FUNCTION_BLOCK Test_TStreamAdd_Read_LINT EXTENDS T_UnitTestBase
VAR
    Stream  : T_Stream(StreamLength := 2);
    ArgType : E_ArgTypeId := E_ArgTypeId.Type_LINT;
END_VAR

METHOD  Init
VAR_INPUT
END_VAR
END_METHOD

{attribute 'analysis' := '-33'} // inhibit unused variable warning
METHOD RunTest
Stream.Init(2);

// add a LINT...
Stream.SetNextArgTypeId(ArgType);
Stream.Add_LINT(123456789);

Stream.SetReadPosition(0);

// check next arg type is correct...
AssertEquals_INT(Expected     := ArgType,
                           Actual       := Stream.GetNextArgTypeId(),
                           Message := 'Stream.GetNextArgTypeId()');

// check next value...	
AssertEquals_LINT(Expected     := 123456789,
                            Actual       := Stream.Read_LINT(),
                            Message := 'Stream.Read_LINT()');

// check we are at the end of the stream..							
AssertEquals_UDINT(Expected     := Stream.StreamLength,
                             Actual       := Stream.ReadPosition,
                             Message := 'Stream.ReadPosition');

TestCompleted := TRUE;
END_METHOD

END_FUNCTION_BLOCK

(* stored: Version 1.1.0.1, ProductVersion 3.1.4024.12
   POU Test_TStreamAdd_Read_LINT: Id {18e29439-c2df-4006-8e67-0957bbd921ad}, SpecialFunc None
   Method Init: Id {efd46019-bafc-4047-93f7-e0ee07a91bc7}
   Method RunTest: Id {db55a77e-ceb3-49ec-856b-7b972c2d482c} *)
